{attribute 'Tc2GvlVarNames'}
VAR_GLOBAL
	MATH : CONSTANTS_MATH;
	PHYS : CONSTANTS_PHYS;
	LANGUAGE : CONSTANTS_LANGUAGE;
	SETUP : CONSTANTS_SETUP;
	LOCATION : CONSTANTS_LOCATION;
END_VAR

(* stored: Version 1.1.0.1
   GVL Globale_Variablen_2: Id {203ff6f3-87b7-4f7d-968a-47c6c41f8d66} *)
